// TIA Portal V20 export
// export: Created 2025-09-12T17:57:00.0000000Z, ExportSetting WithDefaults
TYPE "UDT200_EM_Cooling"
   STRUCT
      CHW_Freeze_Stat_DI : Bool;   // Digital Input: Freeze-stat on chilled water coil (`True` = Fault).
      CHW_Valve_Fdbk_AI : Real;   // Analog Input: Chilled water valve position feedback (0-100%).
      CHW_Valve_Cmd_AO : Real;   // Analog Output: Chilled water valve position command (0-100%).
      CHW_Freeze_Alm : Bool;   // Alarm: Chilled water coil freeze-stat has tripped.
      Valve_Failure_Alm : Bool;   // Alarm: `True` if valve command and feedback do not match.
   END_STRUCT;
END_TYPE
